SUBAPPLICATION Uebung_053 (* DigitalInput_I1-_I4 auf DigitalOutput_Q1-_Q4 *)
  (* Standard: 61499-2 *)
  (* Version 1.0, 2023-10-23, franz *)
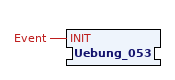
  EVENT_INPUT
    INIT;
  END_EVENT
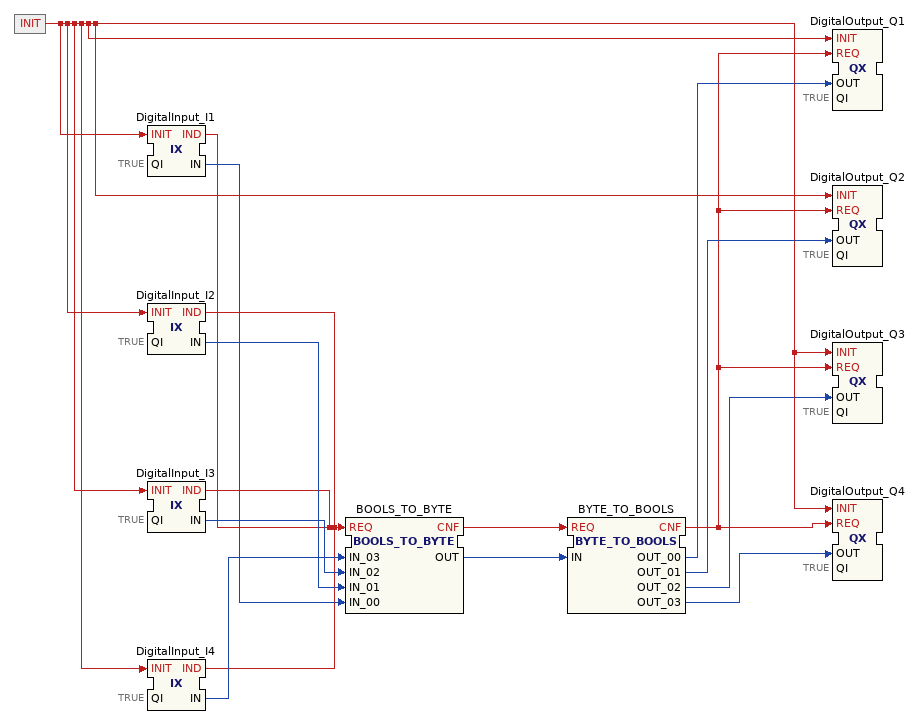
  FBS
    DigitalOutput_Q1 : QX(QI := TRUE);
    DigitalInput_I1 : IX(QI := TRUE);
    DigitalOutput_Q2 : QX(QI := TRUE);
    DigitalInput_I2 : IX(QI := TRUE);
    DigitalOutput_Q3 : QX(QI := TRUE);
    DigitalInput_I3 : IX(QI := TRUE);
    DigitalOutput_Q4 : QX(QI := TRUE);
    DigitalInput_I4 : IX(QI := TRUE);
    BOOLS_TO_BYTE : BOOLS_TO_BYTE;
    BYTE_TO_BOOLS : BYTE_TO_BOOLS;
  END_FBS
  EVENT_CONNECTIONS
    INIT TO DigitalInput_I1.INIT;
    INIT TO DigitalInput_I2.INIT;
    INIT TO DigitalInput_I3.INIT;
    INIT TO DigitalInput_I4.INIT;
    INIT TO DigitalOutput_Q1.INIT;
    INIT TO DigitalOutput_Q2.INIT;
    INIT TO DigitalOutput_Q3.INIT;
    INIT TO DigitalOutput_Q4.INIT;
    BOOLS_TO_BYTE.CNF TO BYTE_TO_BOOLS.REQ;
    DigitalInput_I1.IND TO BOOLS_TO_BYTE.REQ;
    DigitalInput_I2.IND TO BOOLS_TO_BYTE.REQ;
    DigitalInput_I3.IND TO BOOLS_TO_BYTE.REQ;
    DigitalInput_I4.IND TO BOOLS_TO_BYTE.REQ;
    BYTE_TO_BOOLS.CNF TO DigitalOutput_Q1.REQ;
    BYTE_TO_BOOLS.CNF TO DigitalOutput_Q2.REQ;
    BYTE_TO_BOOLS.CNF TO DigitalOutput_Q3.REQ;
    BYTE_TO_BOOLS.CNF TO DigitalOutput_Q4.REQ;
  END_CONNECTIONS
  DATA_CONNECTIONS
    BOOLS_TO_BYTE.OUT TO BYTE_TO_BOOLS.IN;
    BYTE_TO_BOOLS.OUT_00 TO DigitalOutput_Q1.OUT;
    BYTE_TO_BOOLS.OUT_01 TO DigitalOutput_Q2.OUT;
    BYTE_TO_BOOLS.OUT_02 TO DigitalOutput_Q3.OUT;
    BYTE_TO_BOOLS.OUT_03 TO DigitalOutput_Q4.OUT;
    DigitalInput_I4.IN TO BOOLS_TO_BYTE.IN_03;
    DigitalInput_I3.IN TO BOOLS_TO_BYTE.IN_02;
    DigitalInput_I2.IN TO BOOLS_TO_BYTE.IN_01;
    DigitalInput_I1.IN TO BOOLS_TO_BYTE.IN_00;
  END_CONNECTIONS
END_SUBAPPLICATION
